// TIA Portal V20 export
DATA_BLOCK "InstGetSinaAlarms"   // DB74
AUTHOR : Siemens Digital Industries
FAMILY : LAF
NAME : LAF_GetSinaAlarms
VERSION : 1.1
// stored: InstanceOfName LAF_GetSinaAlarms, InstanceOfType FB
"LAF_GetSinaAlarms"
   // VAR_INPUT
   //    enable : Bool := TRUE;
   // END_VAR
   // VAR_OUTPUT
   //    valid { ExternalWritable := 'False'} : Bool := FALSE;
   //    busy { ExternalWritable := 'False'} : Bool := FALSE;
   //    error { ExternalWritable := 'False'} : Bool := FALSE;
   //    status { ExternalWritable := 'False'} : Word := 16#7000;
   //    diagnostics { ExternalWritable := 'False'} : "LAF_typeDiagnostics";
   //    statusWriteRecord { ExternalWritable := 'False'} : DWord := 16#0000_0000;
   //    statusReadRecord { ExternalWritable := 'False'} : DWord := 16#0000_0000;
   // END_VAR
   // VAR_IN_OUT
   //    configuration : Array[*] of "LAF_typeDriveDiagConfig";
   //    moduleInterface : "LAF_typeDriveDiagInterfaceHmi";
   // END_VAR
   // VAR
   //    statInternal { ExternalAccessible := 'False'; ExternalVisible := 'False'; ExternalWritable := 'False'} : Struct
   //       enablePrevious : Bool := FALSE;
   //       valid : Bool := FALSE;
   //       busy : Bool := FALSE;
   //       error : Bool := FALSE;
   //       errorUserCleared : Bool := FALSE;
   //       errorAutoCleared : Bool := FALSE;
   //       disablingCompleted : Bool := FALSE;
   //       diagnostics : "LAF_typeDiagnostics";
   //       emptyDiagnostics : "LAF_typeDiagnostics";
   //    END_STRUCT;
   //    statMainState { ExternalAccessible := 'False'; ExternalVisible := 'False'; ExternalWritable := 'False'} : DInt := 0;
   //    statArrayMin { ExternalAccessible := 'False'; ExternalVisible := 'False'; ExternalWritable := 'False'} : DInt := 0;
   //    statArrayMax { ExternalAccessible := 'False'; ExternalVisible := 'False'; ExternalWritable := 'False'} : DInt := 0;
   //    instWriteRecord { ExternalAccessible := 'False'; ExternalVisible := 'False'; ExternalWritable := 'False'} : WRREC;
   //    instReadRecord { ExternalAccessible := 'False'; ExternalVisible := 'False'; ExternalWritable := 'False'} : RDREC;
   //    statWriteReq { ExternalAccessible := 'False'; ExternalVisible := 'False'; ExternalWritable := 'False'} : Struct
   //       header : Struct
   //          reqRef : Byte := 16#00;
   //          reqID : Byte := 16#00;
   //          axis : Byte := 16#01;
   //          noPara : Byte := 16#01;
   //       END_STRUCT;
   //       data : Array[0..235] of Byte;
   //    END_STRUCT;
   //    statReadReq { ExternalAccessible := 'False'; ExternalVisible := 'False'; ExternalWritable := 'False'} : Struct
   //       header : Struct
   //          reqRef : Byte := 16#00;
   //          reqID : Byte := 16#00;
   //          axis : Byte := 16#01;
   //          noPara : Byte := 16#01;
   //       END_STRUCT;
   //       data : Array[0..235] of Byte;
   //    END_STRUCT;
   //    instActTimer { ExternalAccessible := 'False'; ExternalVisible := 'False'; ExternalWritable := 'False'} : IEC_TIMER;
   //    instReqTimer { ExternalAccessible := 'False'; ExternalVisible := 'False'; ExternalWritable := 'False'} : IEC_TIMER;
   //    statDataTransRun { ExternalAccessible := 'False'; ExternalVisible := 'False'; ExternalWritable := 'False'} : Bool := FALSE;
   //    statWriteReqSet { ExternalAccessible := 'False'; ExternalVisible := 'False'; ExternalWritable := 'False'} : Bool := FALSE;
   //    statActTimerIn { ExternalAccessible := 'False'; ExternalVisible := 'False'; ExternalWritable := 'False'} : Bool := FALSE;
   //    statPrevTimeValue { ExternalAccessible := 'False'; ExternalVisible := 'False'; ExternalWritable := 'False'} : Time := T#0MS;
   //    statActTimerValueAct { ExternalAccessible := 'False'; ExternalVisible := 'False'; ExternalWritable := 'False'} : Time := T#0MS;
   //    statActTimerValueReq { ExternalAccessible := 'False'; ExternalVisible := 'False'; ExternalWritable := 'False'} : Time := T#0MS;
   //    statPrevDriveIndex { ExternalAccessible := 'False'; ExternalVisible := 'False'; ExternalWritable := 'False'} : DInt := 0;
   // END_VAR
BEGIN
   diagnostics.status := 16#0000;
   diagnostics.subfunctionStatus := 16#0000;
   diagnostics.stateNumber := 0;
   statInternal.diagnostics.status := 16#7000;
   statInternal.diagnostics.subfunctionStatus := 16#0000;
   statInternal.diagnostics.stateNumber := 0;
   statInternal.emptyDiagnostics.status := 16#7000;
   statInternal.emptyDiagnostics.subfunctionStatus := 16#0000;
   statInternal.emptyDiagnostics.stateNumber := 0;
   instWriteRecord.REQ := FALSE;
   instWriteRecord.ID := 0;
   instWriteRecord.INDEX := 0;
   instWriteRecord.LEN := 0;
   instWriteRecord.DONE := FALSE;
   instWriteRecord.BUSY := FALSE;
   instWriteRecord.ERROR := FALSE;
   instWriteRecord.STATUS := 16#0000_0000;
   instReadRecord.REQ := FALSE;
   instReadRecord.ID := 0;
   instReadRecord.INDEX := 0;
   instReadRecord.MLEN := 0;
   instReadRecord.VALID := FALSE;
   instReadRecord.BUSY := FALSE;
   instReadRecord.ERROR := FALSE;
   instReadRecord.STATUS := 16#0000_0000;
   instReadRecord.LEN := 0;
   statWriteReq.data[0..235] := 16#00;
   statReadReq.data[0..235] := 16#00;
   instActTimer.PT := T#0MS;
   instActTimer.IN := FALSE;
   instReqTimer.PT := T#0MS;
   instReqTimer.IN := FALSE;
END_DATA_BLOCK
